TYPE ST_Setpoints_Base :
STRUCT
	RequiredChargedV : REAL := 12;
	TotalCapacitance : REAL := 10; //uF - LOCAL ONLY, NOT FROM MAIN PLC - LoadCapacitance
	PSratedV		 : REAL := 50;
	wLCA			 : BOOL := TRUE;
	NumOfCharger	 : INT := 1;
	e_ChargerType		 : E_ChargerType;
END_STRUCT
END_TYPE

(* stored: Version 1.1.0.1, ProductVersion 3.1.4024.11
   DUT ST_Setpoints_Base: Id {0a95a6b7-b17b-4842-b185-de1cd9ac09f2} *)
